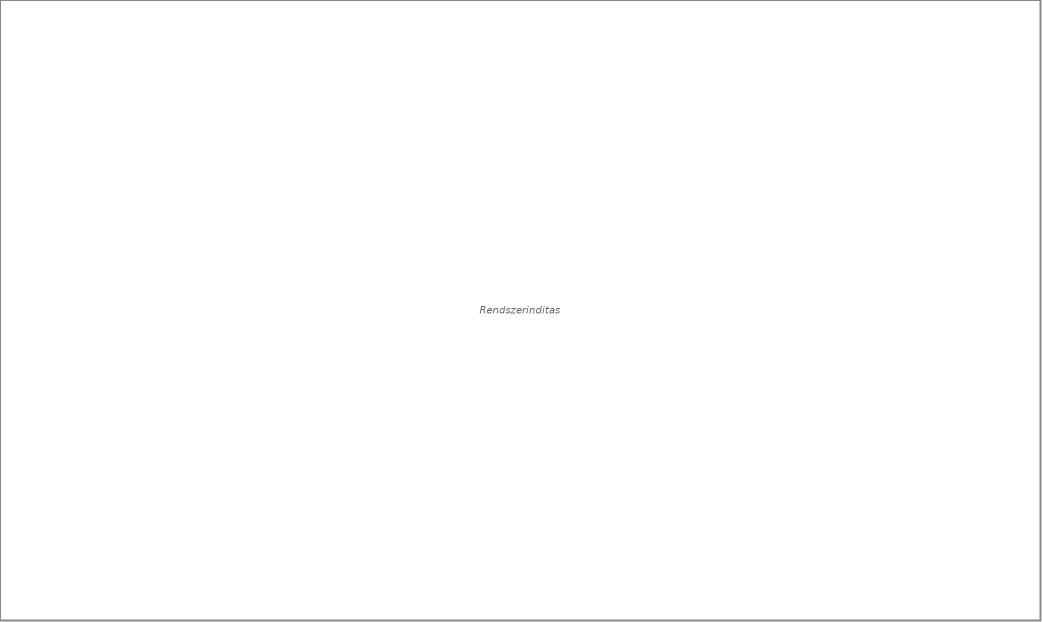
VISUALIZATION Szerviz  // 1042x622
    TabControl (0,0 1040x620), frame switch variable: GVL.iSzervizLapozo
        shows Rendszerinditas()
        shows Behelyezes()
        shows Tengelyek()
        shows Hajlitok()
        shows Hegesztok()
        shows Robot()
        shows NTC_szerviz()
        shows Kappe_pres()
        shows Vegmero()
        shows Lezer()
        shows Kodolvaso()
        shows Himba()
        shows Kamera_Pt()
        [0]: TabTitle=Rendszer
        [1]: TabTitle=Behelyezés
        [2]: TabTitle=Tengelyek
        [3]: TabTitle=Hajlítók
        [4]: TabTitle=Hegesztés
        [5]: TabTitle=Robot
        [6]: TabTitle=NTC vágó
        [7]: TabTitle=Kappe prés
        [8]: TabTitle=Végmérö
        [9]: TabTitle=Lézer
        [10]: TabTitle=Kódolvasó
        [11]: TabTitle=Himba
        [12]: TabTitle=Kamera Pt
END_VISUALIZATION

(* stored: Version 1.1.0.1, ProductVersion 3.1.4024.11
   Visu Szerviz: Id {cd407fe5-0495-4eaa-83db-1d105dd36867} *)
